TYPE ST_SV_Zustand :
STRUCT
	Stellung_Anford		: BOOL;
	Stellung_Soll		: BOOL;
	Stellung			: BOOL;

	Freigabe			: BOOL;
	Freigabe_Deakt		: BOOL;
	Freigabe_Code		: WORD;

	Stoerung			: BOOL;
	Stoerung_Code		: WORD;

	Warnung				: BOOL;
	Warnung_Code		: WORD;

	Status				: SINT;

	Stellungwechsel01	: BOOL;
	Stellungwechsel10	: BOOL;

	Quittierung			: BOOL;

END_STRUCT
END_TYPE

(* stored: Version 1.1.0.1, ProductVersion 3.1.4024.9
   DUT ST_SV_Zustand: Id {43fb4584-049c-408d-a0f1-81c793a80a32} *)
